{attribute 'linkalways'} 
{attribute 'no_explicit_call' := 'This FB is a CLASS and must be accessed using methods or properties'}
{attribute 'enable_dynamic_creation'}
FUNCTION_BLOCK QueueChangedEvent EXTENDS QueueEvent IMPLEMENTS I_QueueChangedEvent

END_FUNCTION_BLOCK

(* stored: Version 1.1.0.1, ProductVersion 3.1.4024.12
   POU QueueChangedEvent: Id {ebe0a914-8727-42fe-a3fc-01c959025295}, SpecialFunc None *)
